FUNCTION_BLOCK FB_ControlElement_HMI EXTENDS FB_BaseControlElement_HMI IMPLEMENTS ITF_ControlElement_HMI
VAR
	itfControlElementConnector			: ITF_ControlElement_HMI_Connector;
	refstControlElementData				: REFERENCE TO ST_ControlElement_HMI;
	
	itfComponent1						: ITF_Component_HMI;
	itfComponent2						: ITF_Component_HMI;
END_VAR

METHOD FB_init : BOOL
VAR_INPUT
	bInitRetains : BOOL; // if TRUE, the retain variables are initialized (warm start / cold start)
	bInCopyCode : BOOL;  // if TRUE, the instance afterwards gets moved into the copy code (online change)
	itfBaseLoggerConnector				: ITF_BaseLogger_HMI_Connector;	//bezpośredni łącznik do logera
	itfControlElementConnector			: ITF_ControlElement_HMI_Init;
	itfComponent1						: ITF_Component_HMI;
	itfComponent2						: ITF_Component_HMI;
END_VAR
//Przypisanie do elementu który własnie stworzyliśmy
THIS^.itfControlElementConnector		:= itfControlElementConnector;
//Przypisanie do elementów z biblioteki
THIS^.itfBaseLoggerElementConnector		:= itfControlElementConnector;
THIS^.itfBaseComponentConnector			:= itfControlElementConnector;
THIS^.itfBaseControlElementConnector	:= itfControlElementConnector;
//
THIS^.itfBaseLoggerConnector			:= itfBaseLoggerConnector;
//
THIS^.itfComponent1						:= itfComponent1;
THIS^.AddComponent (itfComponentHMI		:= itfComponent1);
THIS^.itfComponent2						:= itfComponent2;
this^.AddComponent (itfComponentHMI		:= itfComponent2);

IF (THIS^.itfControlElementConnector <> 0 AND
	THIS^.itfBaseLoggerElementConnector <> 0 AND
	THIS^.itfBaseComponentConnector	<> 0 AND
	THIS^.itfBaseControlElementConnector <> 0 AND
	THIS^.itfBaseLoggerConnector <> 0) THEN
	THIS^.bIsInit						:= TRUE;
END_IF
END_METHOD

METHOD LinkControlElementData : BOOL
VAR_INPUT
	stData				: reference to ST_ControlElement_HMI_Link;
END_VAR
THIS^.refstControlElementData			REF= stData.stControlElement;	//ta zmienna powstaje w elemencie 

THIS^.refstBaseLoggerElementDataHMI		REF= stData.stBaseLoggerElement;	//zmienne z biblioteki ale dopiero tu je moge przypisać 
THIS^.refstBaseComponentDataHMI			REF= stData.stBaseComponent;
THIS^.refstBaseControlElementDataHMI	REF= stData.stBaseControlElement;

THIS^.itfComponent1.LinkComponentData (stData := stData.stComponent1);	//przekazanie danych do elementu podrzędnego np do czujnika
THIS^.itfComponent2.LinkComponentData (stData := stData.stComponent2);

THIS^.CreateLinkToEventsMemory ();	//wywołanie metody linkującą poamięc zgłoszęń

IF (__ISVALIDREF (THIS^.refstControlElementData) AND this^.IsLinkedReferences ()) THEN
	THIS^.bIsValidData		:= TRUE;
	LinkControlElementData	:= TRUE;
END_IF
END_METHOD

END_FUNCTION_BLOCK

(* stored: Version 1.1.0.1, ProductVersion 3.1.4024.15
   POU FB_ControlElement_HMI: Id {6ebe5482-b91b-4d08-bc26-129cdd0cb96c}, SpecialFunc None
   Folder ITF_ControlElement_HMI: Id {4058a596-c262-4ce5-adbb-2422ae7eb30c}
   Method FB_init: Id {b9738a13-18ea-4753-90b7-8525f5e660e5}
   Method LinkControlElementData: Id {9ee2bb6f-ad99-45ad-b84c-15e014e2b842} *)
